TYPE typDMXOutput :
STRUCT
	byStatValue			: BYTE;
	fFnGeneratorVal		: LREAL;
END_STRUCT
END_TYPE

(* stored: Version 1.1.0.1, ProductVersion 3.1.4024.6
   DUT typDMXOutput: Id {b5532f2b-075e-4f4f-8c62-43bc1be2ce13} *)
